FUNCTION_BLOCK T_RoboConnect_SetAnalogOutput_TimeoutFails EXTENDS T_UnitTestBase
VAR
  robot : I_RoboConnect;
  timeOutTimer : TON;
  targetAO : UINT;
  myTestState, prevState :
    (INIT,
    ARRANGE,
    ACT,
    ASSERT) := INIT;
  expected, actual : BOOL;
  counter : UINT;
  returnedTask : I_Task;
END_VAR

CASE myTestState OF
  INIT:
    StateChanged();
    myTestState := ARRANGE;

  ARRANGE:
    IF StateChanged() THEN
      expected := TRUE;
      robot.Connect();
    END_IF

    IF robot.Connected THEN
      myTestState := ACT;
    END_IF

  ACT:
    robot.SetDigitalOutput(targetAO,TRUE, task => returnedTask);
    myTestState := ASSERT;

  ASSERT:
    IF timeOutTimer.Q THEN
      actual := returnedTask.Timeout;
      assertion.AssertEquals_BOOL(expected, actual, 'actual := returnedTask.Timeout');
      TestFinished();
      myTestState := INIT;

    END_IF

END_CASE

robot.CyclicLogic();
timeOutTimer(IN := myTestState = ASSERT);

METHOD FB_init : BOOL
VAR_INPUT
  bInitRetains : BOOL; // if TRUE, the retain variables are initialized (warm start / cold start)
  bInCopyCode : BOOL; // if TRUE, the instance afterwards gets moved into the copy code (online change)
  TestSuite : tcl_SimpleUnitTestLibrary.I_TestSuite;
  robot : I_TcRobot;
  targetAo : UINT;
  timeout : TIME;
END_VAR
THIS^.robot := robot;
THIS^.timeoutTimer.PT := timeout;
THIS^.targetAo := targetAo;
END_METHOD

METHOD PRIVATE StateChanged : BOOL
IF  myTestState = prevState THEN
  RETURN;
END_IF

prevState := myTestState;
StateChanged := TRUE;
END_METHOD

METHOD WaitForCycles : BOOL
VAR_INPUT
  maxCount : UINT;
END_VAR
counter := counter + 1;

IF counter = maxCount THEN
  counter := 0;
  WaitForCycles := TRUE;
END_IF
END_METHOD

END_FUNCTION_BLOCK

(* stored: Version 1.1.0.1
   POU T_TcRobot_SetAnalogOutput_TimeoutFails: Id {33999cfb-aaba-4e4b-8cc4-178f456b901a}, SpecialFunc None
   Method FB_init: Id {4e3d4fd8-68aa-441d-bea0-b1eaa99a0cdb}
   Method StateChanged: Id {729e8e0f-c1ba-495e-bb02-0197cdd74405}
   Method WaitForCycles: Id {635b8f51-c885-4642-a7cb-8ead6bafc957} *)
